FUNCTION_BLOCK FB_TOR_SD EXTENDS FB_TOR_Base
//////////////////
//  Smoke and Fire detection system with Typhoon triggering system. 
//////////////////
VAR_INPUT PERSISTENT
	// Parameters of the Object (instance/model specific) 
	ParamTempoFire :TIME:=T#2S;(*  (s)Tempo before raising an alarm*)
END_VAR

VAR_OUTPUT
	//Child objects
		OUT_FireDetection	: BOOL;
END_VAR

VAR_INPUT
	// I/O Inputs 		                                     				
		
		MesDataExd			: TOR_Standard ;  

END_VAR

VAR
	//M_ALARMMANAGEMENT VARIABLES//
		FB_PermAlarm				: SR ;					// (NA) FB to maintain Fire Alarm even if sensor stop detection (burn) .
		TON_Fire					: TON ; 
 
	//M_STATEMANAGER VARIABLES//
		
END_VAR

METHOD M_AlarmManagement
//////////////////
// Manages Smoke detector alarms and warnings
/////////////////

VAR 
	// Method local variables (reinitialized at each cycle) 
	FB_AlarmCodeManager			: FB_AlarmCodeManager ; 
	bTrigDaily 					: BOOL;
END_VAR
// Detection Variables
TON_Fire(IN:= MesDataExd.MesData.MesAlarmState, PT:= ParamTempoFire ) ; 
FB_PermAlarm(SET1 := TON_Fire.Q  , Reset := CmdClearFault_G OR IN_CmdReset_L ); // SR FB for keep fire if burn .

bTrigDaily := (CalLocalTimeStruct.wHour = 10 OR CalLocalTimeStruct.wHour = 16) AND CalLocalTimeStruct.wMinute = 0;

OUT_FireDetection 	:= FB_PermAlarm.Q1;

IF IN_CmdReset_L THEN
	IN_CmdReset_L := FALSE;
END_IF

// ALARM CODE //
	FB_AlarmCodeManager(
		bAlarm1			:= OUT_FireDetection ,  				// Fire Detection		
		bAlarm2			:= bTrigDaily AND OUT_FireDetection,	// Reminder : fire detection still active. 
		bAlarm3			:=FALSE, 								// 
		bAlarm4			:=FALSE, 								// 
		bAlarm5			:=FALSE, 								//
		bAlarm6			:=FALSE,                            	//
		bAlarm7			:=FALSE,                            	//
		bAlarm8			:=FALSE,                            	//
		bAlarm9			:=FALSE,                            	//
		bAlarm10		:=FALSE,                            	//
		bAlarm11		:=FALSE,                            	//
		bAlarm12		:=FALSE,                            	//
		bAlarm13		:=FALSE,                            	//
		bAlarm14		:=FALSE,                            	//
		bAlarm15		:=FALSE,                            	//
		wAlarmCode		=>MesDataExd.MesData.MesAlarmCode );
		
// WARNING CODE //
	FB_AlarmCodeManager(
		bAlarm1			:=FALSE,	  															// 
		bAlarm2			:=FALSE, 																//
		bAlarm3			:=FALSE, 																// 
		bAlarm4			:=FALSE, 																// 
		bAlarm5			:=FALSE, 																// 
		bAlarm6			:=FALSE,                                                                //
		bAlarm7			:=FALSE,                                                                //
		bAlarm8			:=FALSE,                                                                //
		bAlarm9			:=FALSE,                                                                //
		bAlarm10		:=FALSE,                                                                //
		bAlarm11		:=FALSE,                                                                //
		bAlarm12		:=FALSE,                                                                //
		bAlarm13		:=FALSE,                                                                //
		bAlarm14		:=FALSE,                                                                //
		bAlarm15		:=FALSE,                                                                //
		wAlarmCode			=>MesDataExd.MesData.MesWarningCode);
		
// EVENT CODE //
	FB_AlarmCodeManager(
		bAlarm1			:= IN_MesState1_IO, 		// First sensor is ON
		bAlarm2			:= IN_MesState2_IO, 		// Second sensor is ON
		bAlarm3			:= FALSE, 					// 		
		bAlarm4			:= FALSE, 					// 
		bAlarm5			:= FALSE, 					//
		bAlarm6			:= FALSE,                   //
		bAlarm7			:= FALSE,                   //
		bAlarm8			:= FALSE,                   //
		bAlarm9			:= FALSE,                   //
		bAlarm10		:= FALSE,                   //
		bAlarm11		:= FALSE,                   //
		bAlarm12		:= FALSE,                   //
		bAlarm13		:= FALSE,                   //
		bAlarm14		:= FALSE,                   //
		bAlarm15		:= FALSE,                   //
		wAlarmCode		=>MesDataExd.MesData.MesEventCode);
END_METHOD

METHOD M_Execute
//////////////////
//  Method Calls 
/////////////////

VAR 
	// Method local variables (reinitialized at each cycle) 

END_VAR

	IF ParamNbSensors = 9 THEN // Use of contactor bi-stable No and NC
		IN_MesState2_IO := NOT IN_MesState2_IO;
	END_IF
SUPER^.M_Execute() ;
END_METHOD

METHOD M_StateManager
//////////////////
// Detect when fire occurs
/////////////////

VAR 
	// Method local variables (reinitialized at each cycle)
 	MesStateInterm1 : BOOL;
	MesStateInterm2 : BOOL;
END_VAR

IF ParamCableCutSecurity THEN
	MesStateInterm1 := NOT IN_MesState1_IO ; 
	MesStateInterm2 := NOT IN_MesState2_IO ; 
ELSE 
	MesStateInterm1 := IN_MesState1_IO;
	MesStateInterm2 := IN_MesState2_IO;
END_IF

IF ParamNbSensors = 1 THEN 
	MesStateInterm2 := MesStateInterm1 ;
END_IF

IF ParamAtleastOne THEN 
MesDataExd.MesData.MesAlarmState := MesStateInterm1 OR MesStateInterm2 ; 
ELSE
MesDataExd.MesData.MesAlarmState := MesStateInterm1 AND MesStateInterm2 ; 
END_IF

R_TRIGAlarm(CLK:= MesDataExd.MesData.MesAlarmState ) ; 
IF R_TRIGAlarm.Q THEN
	MesCountAlarm :=  MIN(MesCountAlarm + 1 ,4294967295 ) ; 
ELSIF IN_ResetCounter THEN 
	MesCountAlarm := 0 ; 
END_IF

MesDataExd.MesData.MesCountAlarm	:= MesCountAlarm ;
END_METHOD

END_FUNCTION_BLOCK

(* stored: Version 1.1.0.1, ProductVersion 3.1.4024.14
   POU FB_TOR_SD: Id {90dc2fe8-b2b7-433d-ae09-aa441c1a15e4}, SpecialFunc None
   Method M_AlarmManagement: Id {bf04f165-0833-4ee3-9edc-1ee259c1678c}
   Method M_Execute: Id {8a526882-db39-4f89-9bc6-69e135744eec}
   Method M_StateManager: Id {6cbd8098-f8f8-4b44-905c-5200dc0f0cb4} *)
